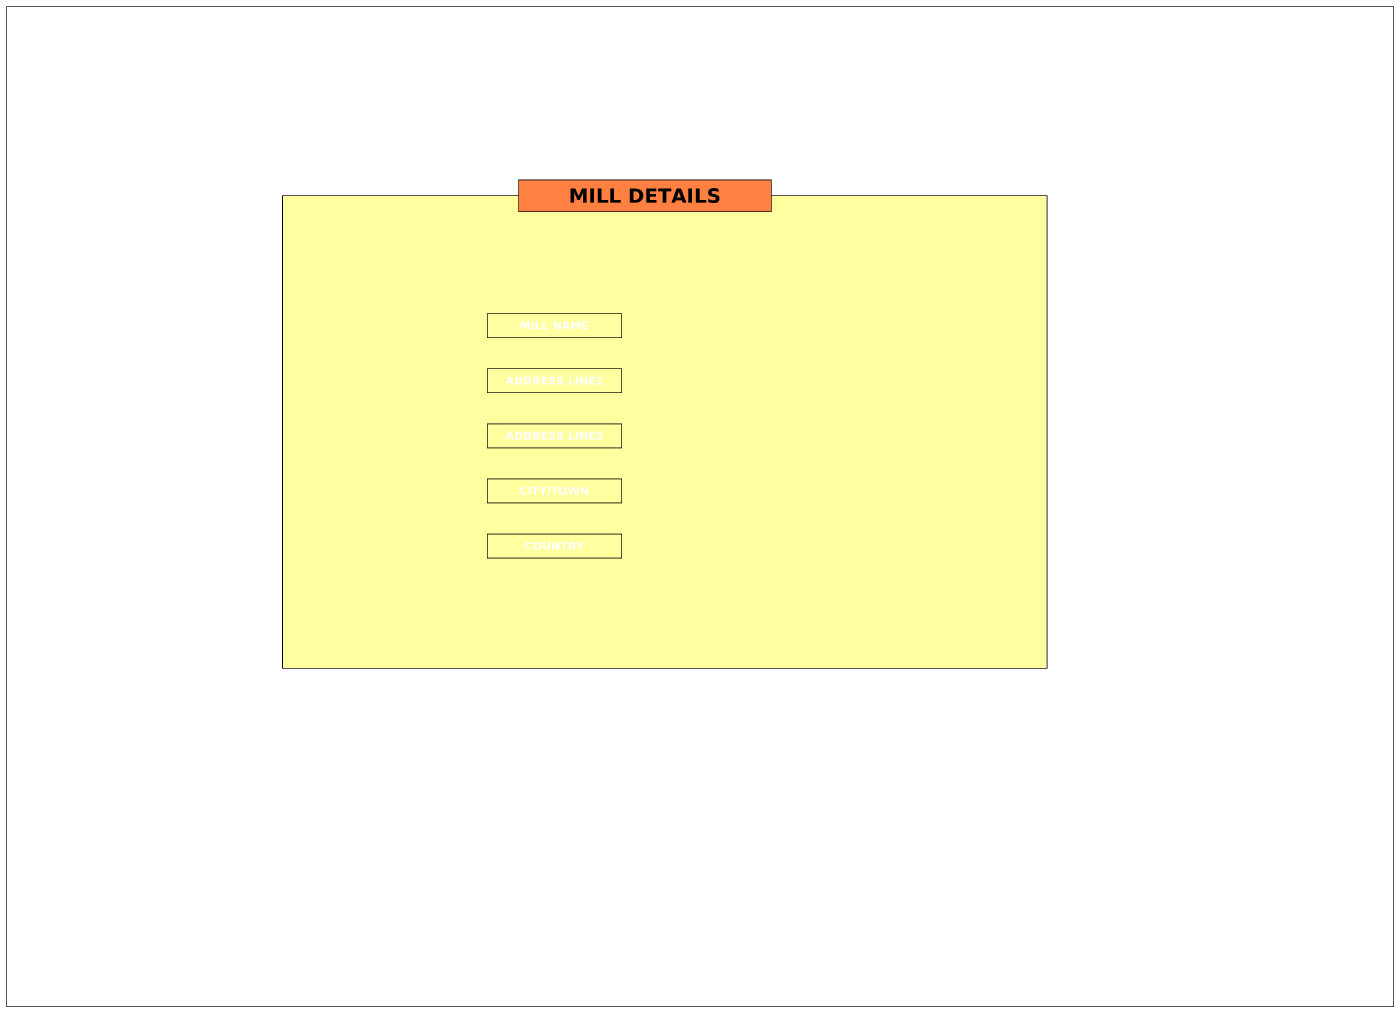
rectangle at (610,390)-(781,421): text "MILL NAME"
rectangle at (610,460)-(781,491): text "ADDRESS LINE1"
rectangle at (610,530)-(781,561): text "ADDRESS LINE2"
rectangle at (610,600)-(781,631): text "CITY/TOWN"
rectangle at (610,670)-(781,701): text "COUNTRY"
rounded rectangle at (650,220)-(971,261): text "MILL DETAILS"
2 more shapes without text or variables
9 elements of other kinds (tables, trends, ...) not read
*)

(* Visualisation MODELS
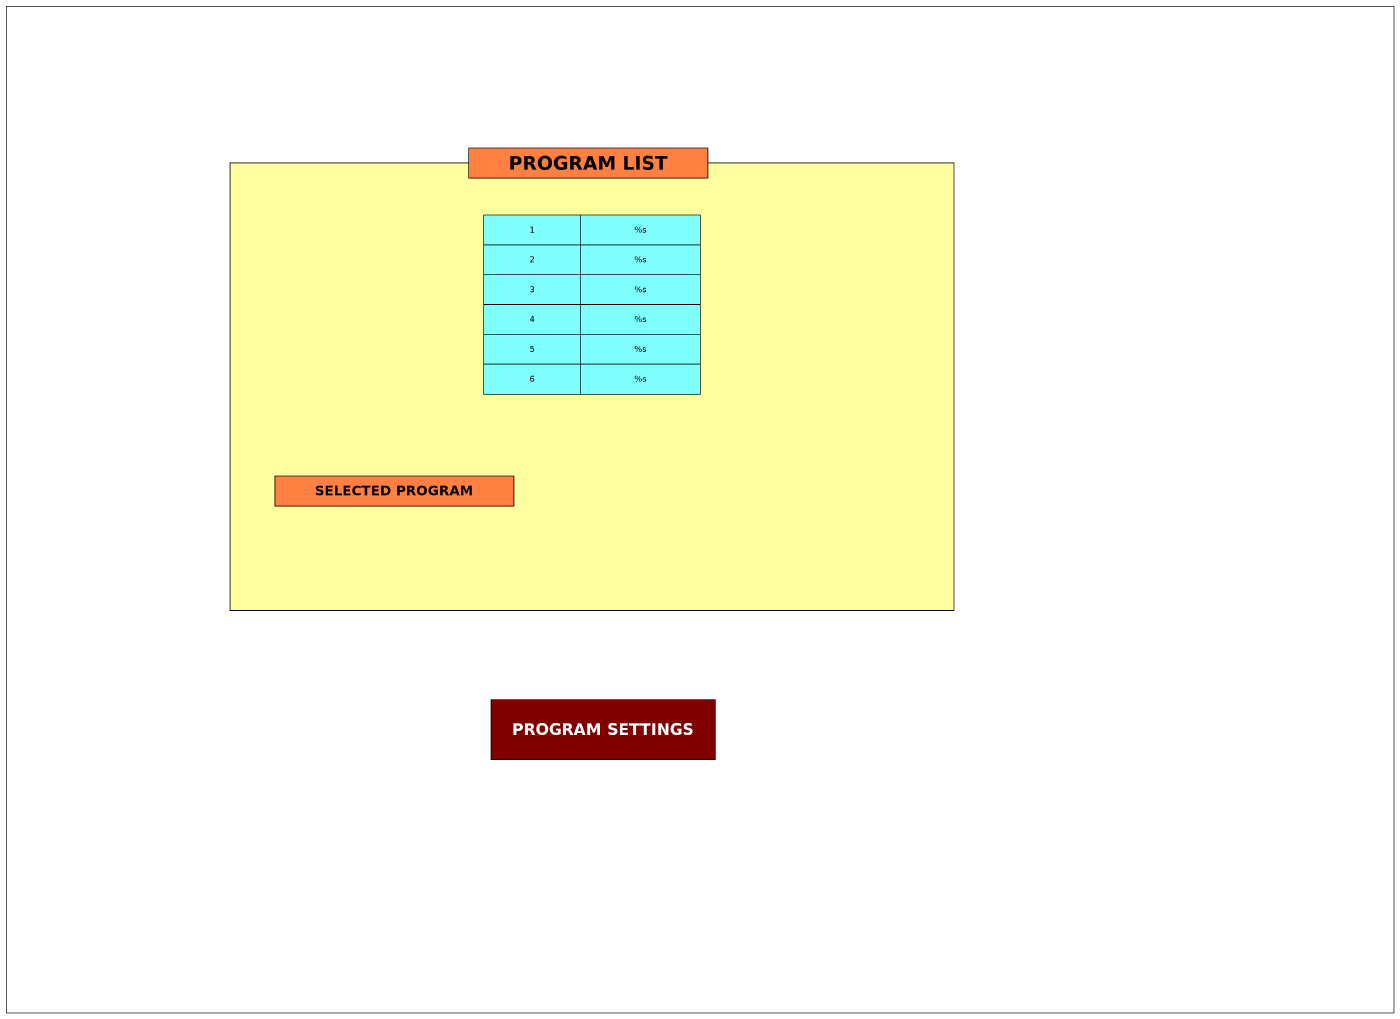
rectangle at (630,280)-(761,321): text "1"; taps bModel1Hmi
rectangle at (760,280)-(921,321): text "%s"; shows PgmNameDis1
rectangle at (630,320)-(761,361): text "2"; taps bModel2Hmi
rectangle at (760,320)-(921,361): text "%s"; shows PgmNameDis2
rectangle at (630,360)-(761,401): text "3"; taps bModel3Hmi
rectangle at (760,360)-(921,401): text "%s"; shows PgmNameDis3
rectangle at (630,400)-(761,441): text "4"; taps bModel4Hmi
rectangle at (760,400)-(921,441): text "%s"; shows PgmNameDis4
rectangle at (630,440)-(761,481): text "5"; taps bModel5Hmi
rectangle at (760,440)-(921,481): text "%s"; shows PgmNameDis5
rectangle at (630,480)-(761,521): text "6"; taps bModel6Hmi
rectangle at (760,480)-(921,521): text "%s"; shows PgmNameDis6
rounded rectangle at (610,190)-(931,231): text "PROGRAM LIST"
rounded rectangle at (350,630)-(671,671): text "SELECTED PROGRAM"
rounded rectangle at (640,930)-(941,1011): text "PROGRAM SETTINGS"; opens PROGRAM_SETTINGS
2 more shapes without text or variables
6 elements of other kinds (tables, trends, ...) not read
*)

(* Visualisation PROGRAM_SETTINGS
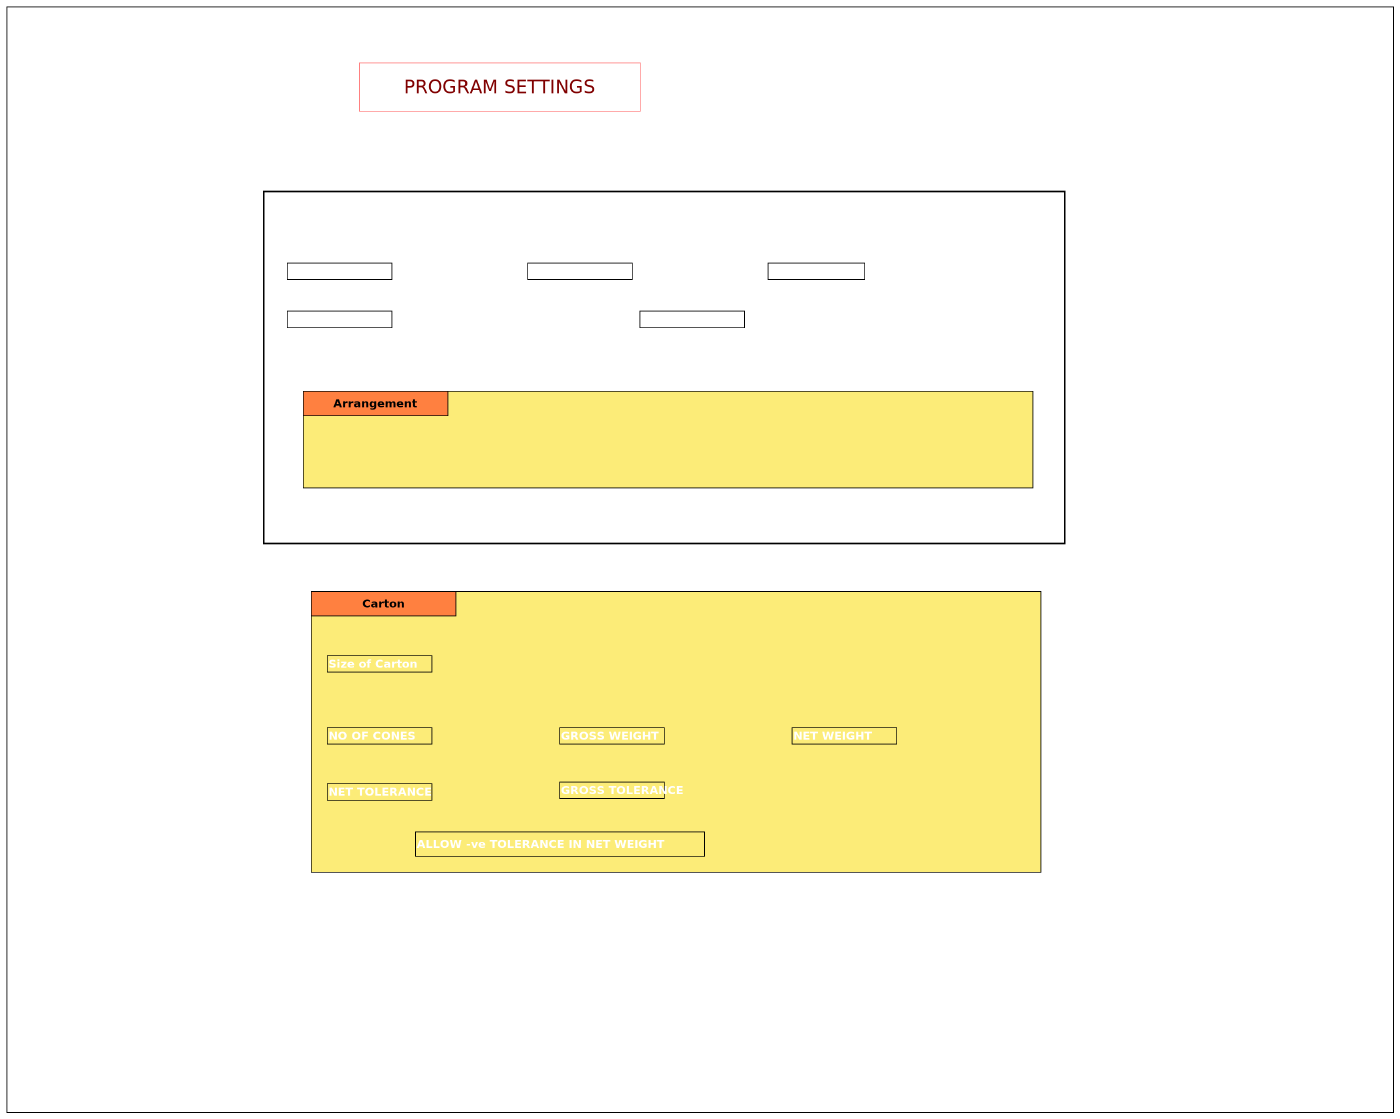
rounded rectangle at (440,0)-(791,61): text "PROGRAM SETTINGS"
rectangle at (380,660)-(561,691): text "Carton"
rounded rectangle at (400,830)-(531,851): text "NO OF CONES"
rounded rectangle at (690,830)-(821,851): text "GROSS WEIGHT"
rounded rectangle at (980,830)-(1111,851): text "NET WEIGHT"
rounded rectangle at (400,900)-(531,921): text "NET TOLERANCE"
rounded rectangle at (690,898)-(821,919): text "GROSS TOLERANCE"
rounded rectangle at (350,250)-(481,271): text "PROGRAM NO"
rounded rectangle at (950,250)-(1071,271): text "DETAILS"
rounded rectangle at (650,250)-(781,271): text "COUNT"
rounded rectangle at (350,310)-(481,331): text "LOT NO"
rounded rectangle at (790,310)-(921,331): text "CARTON NO"
rectangle at (370,410)-(551,441): text "Arrangement"
rounded rectangle at (510,960)-(871,991): text "ALLOW -ve TOLERANCE IN NET WEIGHT"
rounded rectangle at (400,740)-(531,761): text "Size of Carton"
4 more shapes without text or variables
24 elements of other kinds (tables, trends, ...) not read
*)

(* Visualisation RUNNING_STATUS
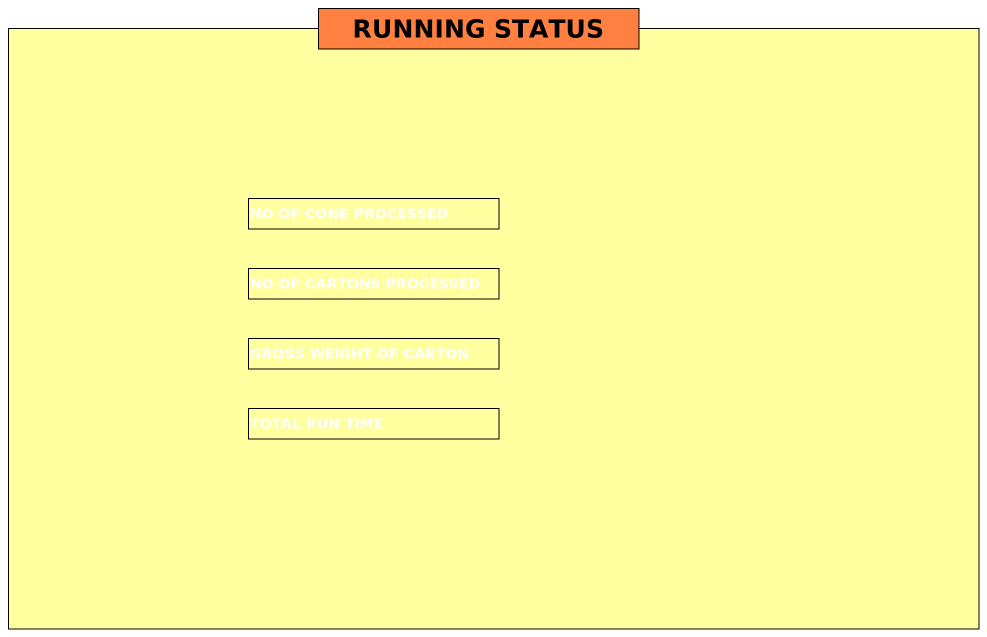
rounded rectangle at (420,280)-(671,311): text "NO OF CONE PROCESSED"
rounded rectangle at (420,350)-(671,381): text "NO OF CARTONS PROCESSED"
rounded rectangle at (420,420)-(671,451): text "GROSS WEIGHT OF CARTON"
rounded rectangle at (420,490)-(671,521): text "TOTAL RUN TIME"
rounded rectangle at (490,90)-(811,131): text "RUNNING STATUS"
1 more shapes without text or variables
7 elements of other kinds (tables, trends, ...) not read
*)

(* Visualisation SERVICE
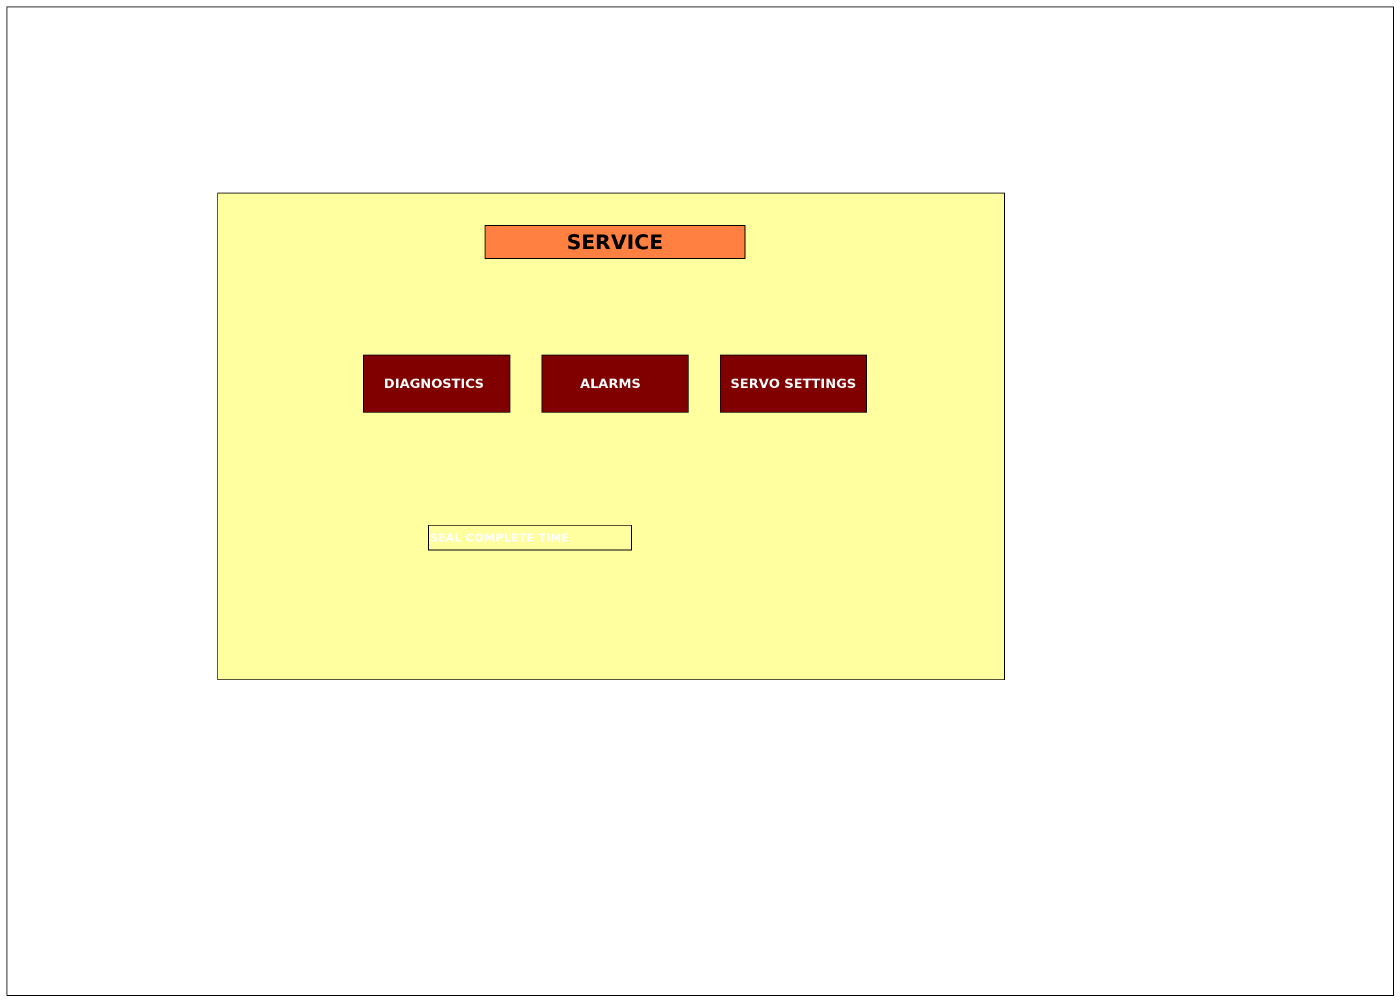
rounded rectangle at (860,430)-(1041,501): text "SERVO SETTINGS"; opens Servo
rounded rectangle at (500,640)-(751,671): text "SEAL COMPLETE TIME"
rounded rectangle at (640,430)-(821,501): text "ALARMS"; opens ALARM
rounded rectangle at (420,430)-(601,501): text "DIAGNOSTICS"; opens DIAGNOSTICS
rounded rectangle at (570,270)-(891,311): text "SERVICE"
2 more shapes without text or variables
4 elements of other kinds (tables, trends, ...) not read
*)

(* Visualisation SERVO
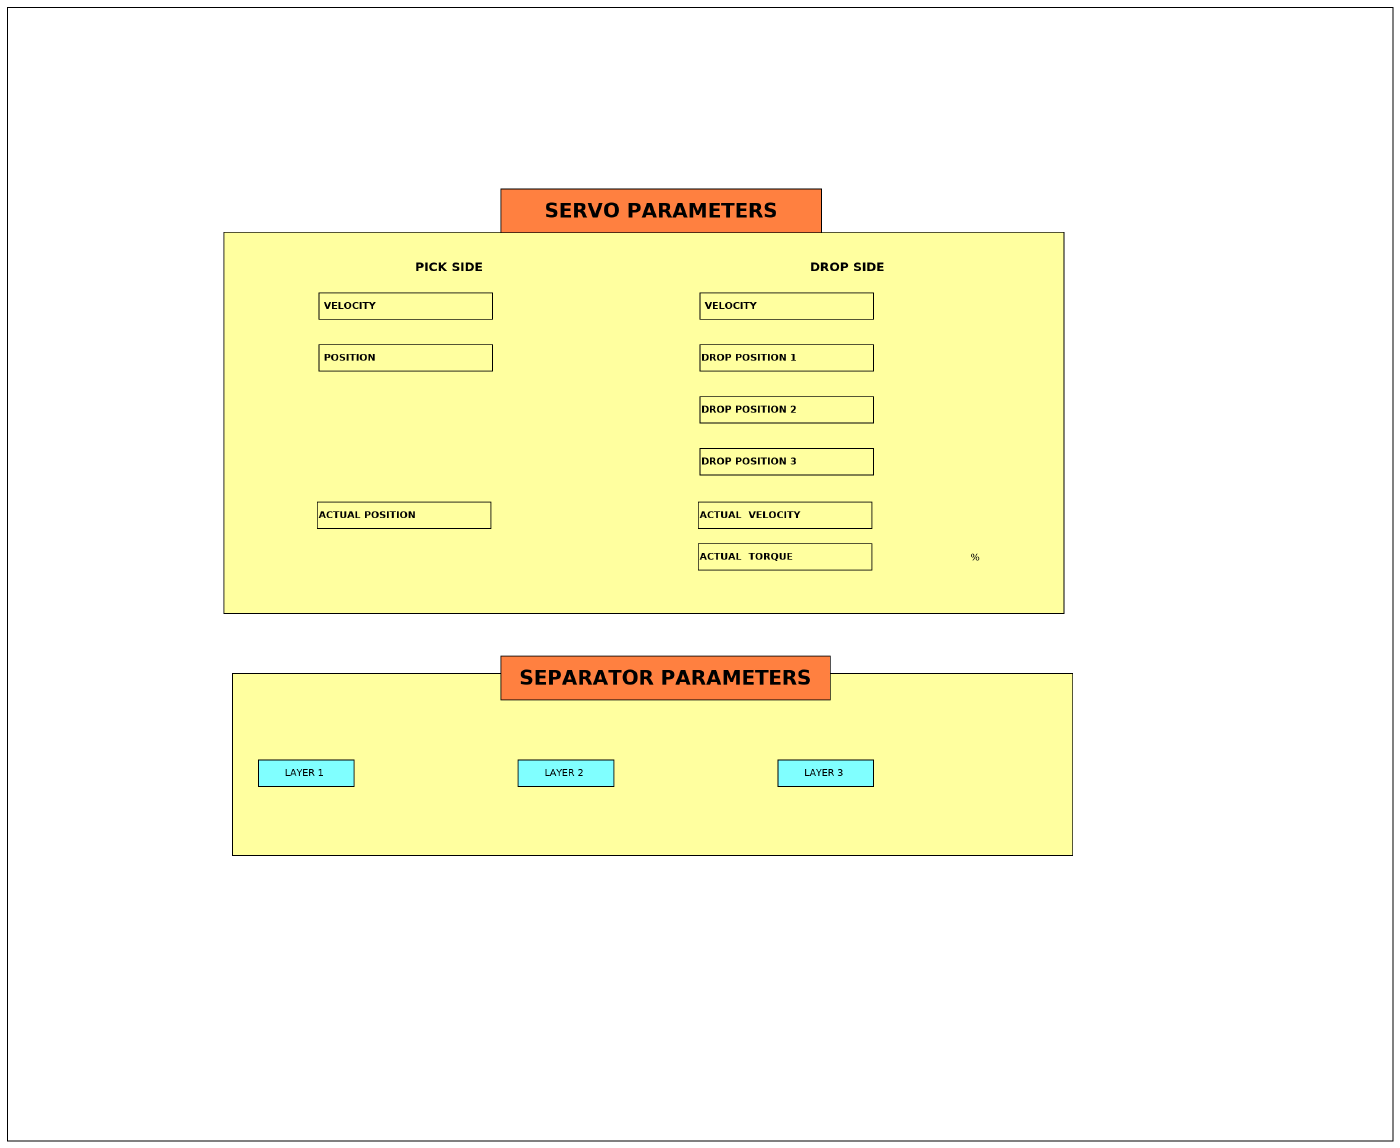
rounded rectangle at (410,230)-(611,271): text "PICK SIDE"
rounded rectangle at (870,230)-(1071,271): text "DROP SIDE"
rounded rectangle at (290,820)-(401,851): text "LAYER 1"
rounded rectangle at (590,820)-(701,851): text "LAYER 2"
rounded rectangle at (890,820)-(1001,851): text "LAYER 3"
rounded rectangle at (570,160)-(941,211): text "SERVO PARAMETERS"
rounded rectangle at (570,700)-(951,751): text "SEPARATOR PARAMETERS"
rounded rectangle at (360,280)-(561,311): text "VELOCITY"
rounded rectangle at (360,340)-(561,371): text "POSITION"
rounded rectangle at (800,280)-(1001,311): text "VELOCITY"
rounded rectangle at (800,340)-(1001,371): text "DROP POSITION 1"
rounded rectangle at (800,400)-(1001,431): text "DROP POSITION 2"
rounded rectangle at (800,460)-(1001,491): text "DROP POSITION 3"
rounded rectangle at (798,522)-(999,553): text "ACTUAL  VELOCITY"
rounded rectangle at (358,522)-(559,553): text "ACTUAL POSITION"
rounded rectangle at (798,570)-(999,601): text "ACTUAL  TORQUE"
rounded rectangle at (1094,570)-(1143,603): text "%"
3 more shapes without text or variables
15 elements of other kinds (tables, trends, ...) not read
*)

(* Visualisation SHIFT
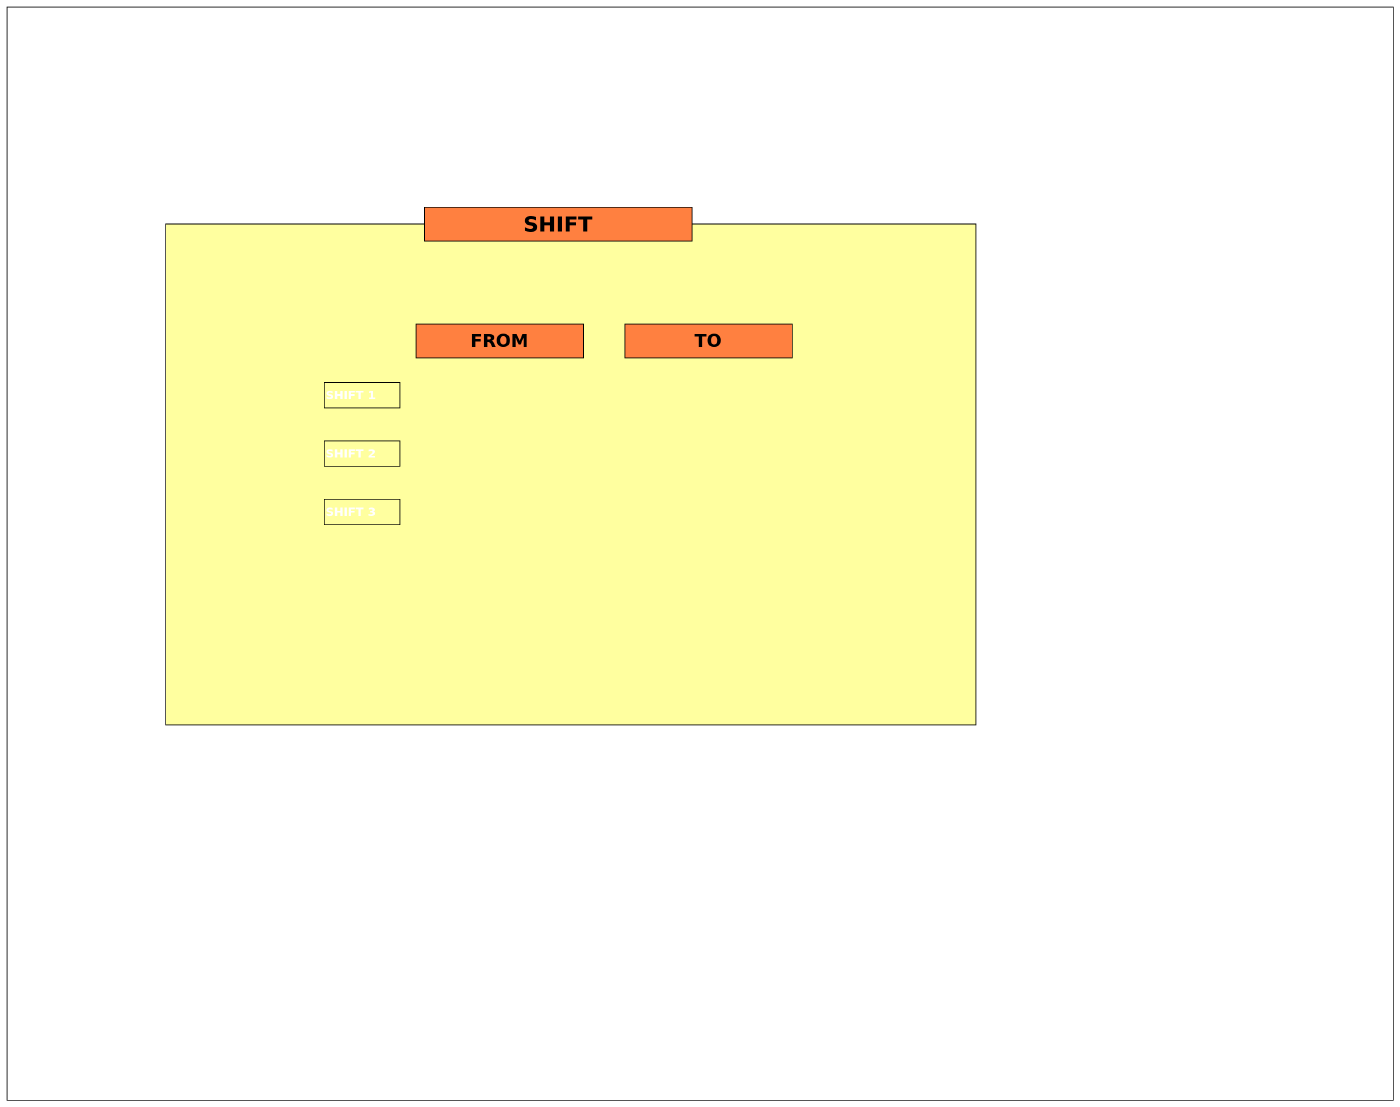
rounded rectangle at (380,450)-(471,481): text "SHIFT 1"
rounded rectangle at (380,520)-(471,551): text "SHIFT 2"
rounded rectangle at (380,590)-(471,621): text "SHIFT 3"
rounded rectangle at (500,240)-(821,281): text "SHIFT"
rounded rectangle at (490,380)-(691,421): text "FROM"
rounded rectangle at (740,380)-(941,421): text "TO"
2 more shapes without text or variables
16 elements of other kinds (tables, trends, ...) not read
*)
